{attribute 'qualified_only'}
VAR_GLOBAL
	alarm_test	: BOOL;
	test		: BOOL;
	RemoteModeSelected : BOOL;

END_VAR

VAR_GLOBAL CONSTANT
	MAX_CSV_ROWS 			: UDINT := 500;
	MAX_CSV_COLUMNS 		: UDINT := 2;
	MAX_CSV_FIELD_LENGTH	: UDINT := 150;
END_VAR

(* stored: Version 1.1.0.1, ProductVersion 3.1.4024.11
   GVL GVL: Id {cc46053f-202c-49b0-8a45-91613fe6626a} *)
